FUNCTION_BLOCK RingTokenHasnotCTL (* Basic Function Block Type *)
  (* Standard: 61499-2 *)
  (* Version 0.2, 2003-12-04, JHC, Rockwell Automation, Renamed for better indexing. *)
  (* Version 0.1, 2002-11-05, JHC, Rockwell Automation, Corrected missing ST element in Algorithm REQ. *)
  (* Version 0.0, 2000-05-30, JHC, Rockwell Automation *)
  (* Compiler header: package fb.rt.cs725; *)
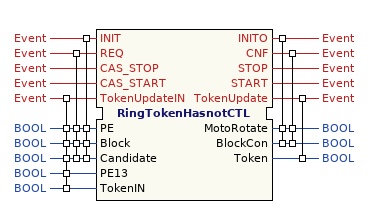
  EVENT_INPUT
    INIT WITH PE, Block, Candidate; (* Initialization Request *)
    REQ WITH PE, Block, Candidate; (* Normal Execution Request *)
    CAS_STOP;
    CAS_START;
    TokenUpdateIN WITH PE, Block, Candidate, PE13, TokenIN;
  END_EVENT
  EVENT_OUTPUT
    INITO WITH MotoRotate, BlockCon; (* Initialization Confirm *)
    CNF WITH MotoRotate, BlockCon; (* Execution Confirmation *)
    STOP;
    START;
    TokenUpdate WITH Token;
  END_EVENT
  VAR_INPUT
    PE : BOOL; (* Input event qualifier *)
    Block : BOOL;
    Candidate : BOOL;
    PE13 : BOOL;
    TokenIN : BOOL;
  END_VAR
  VAR_OUTPUT
    MotoRotate : BOOL; (* Output event qualifier *)
    BlockCon : BOOL;
    Token : BOOL;
  END_VAR
  VAR
    lastPE : BOOL := 1;
    lastBlock : BOOL := 0;
  END_VAR
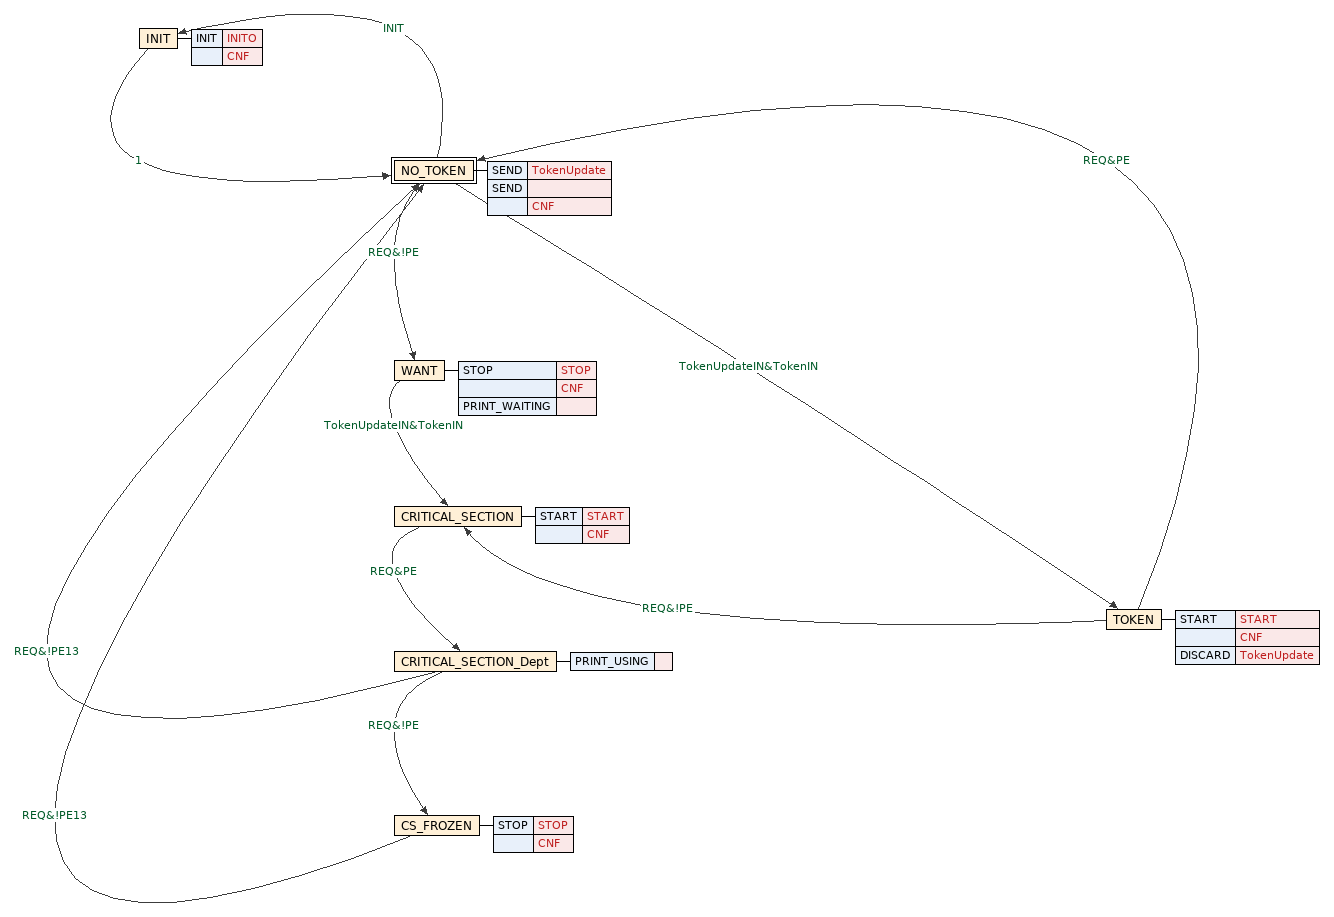
  EC_STATES
    NO_TOKEN : SEND -> TokenUpdate, SEND, -> CNF;
    TOKEN : START -> START, -> CNF, DISCARD -> TokenUpdate;
    INIT : INIT -> INITO, -> CNF;
    CRITICAL_SECTION : START -> START, -> CNF;
    CRITICAL_SECTION_Dept : PRINT_USING;
    CS_FROZEN : STOP -> STOP, -> CNF;
    WANT : STOP -> STOP, -> CNF, PRINT_WAITING;
  END_STATES
  EC_TRANSITIONS
    TOKEN TO NO_TOKEN := REQ&PE;
    NO_TOKEN TO TOKEN := TokenUpdateIN&TokenIN;
    TOKEN TO CRITICAL_SECTION := REQ&!PE;
    CRITICAL_SECTION TO CRITICAL_SECTION_Dept := REQ&PE;
    CRITICAL_SECTION_Dept TO CS_FROZEN := REQ&!PE;
    CRITICAL_SECTION_Dept TO NO_TOKEN := REQ&!PE13;
    CS_FROZEN TO NO_TOKEN := REQ&!PE13;
    WANT TO CRITICAL_SECTION := TokenUpdateIN&TokenIN;
    NO_TOKEN TO WANT := REQ&!PE;
    INIT TO NO_TOKEN := 1;
    NO_TOKEN TO INIT := INIT;
  END_TRANSITIONS
  ALGORITHM INIT IN ST: (* Initialization algorithm *)
MotoRotate := TRUE;
Block := FALSE;
  END_ALGORITHM
  ALGORITHM REQ IN Java: (* Normally executed algorithm *)
if(Candidate.value){
if(lastPE.value!=PE.value){
if(!PE.value){
BlockCon.value=true;
}
 else {
BlockCon.value=false;
}
lastPE.value=PE.value;
}
if(lastBlock.value!=Block.value){
if(Block.value){
STOP.serviceEvent(this);
MotoRotate.value=false;
}
 else {
START.serviceEvent(this);
MotoRotate.value=true;
}
lastBlock.value=Block.value;
}
}
  END_ALGORITHM
  ALGORITHM START IN ST:
MotoRotate:=TRUE;
  END_ALGORITHM
  ALGORITHM STOP IN ST:
MotoRotate := FALSE;
  END_ALGORITHM
  ALGORITHM DISCARD IN Java:
Token.value = false;
  END_ALGORITHM
  ALGORITHM SEND IN Java:
Token.value = true;
  END_ALGORITHM
  ALGORITHM PRINT_WAITING IN Java:
System.out.println(this+" does not have ring token");
  END_ALGORITHM
  ALGORITHM PRINT_USING IN Java:
System.out.println(this+" has Ring Token");
  END_ALGORITHM
END_FUNCTION_BLOCK
